// TIA Portal V16 export
// export: Created 2021-11-12T13:32:49.9949051Z, ExportSetting WithDefaults, DisplayName Totally Integrated Automation Portal, DisplayVersion V16 Update 3, DisplayName TIA Portal Version Control Interface, DisplayVersion V16 Update 2, DisplayName TIA Portal Openness, DisplayVersion V16 Update 3, DisplayName SINAMICS Startdrive Advanced, DisplayVersion V16 Update 5, DisplayName SINAMICS Startdrive G130, G150, S120, S150, SINAMICS MV, S210, DisplayVersion V16 Update 5, DisplayName SINAMICS Startdrive G110M, G120, G120C, G120D, G120P, G115D, DisplayVersion V16 Update 5, DisplayName STEP 7 Professional, DisplayVersion V16 Update 3, DisplayName STEP 7 Safety, DisplayVersion V16, DisplayName WinCC UA Professional, DisplayVersion V16 Update 3
DATA_BLOCK "HMI_CMD_310"   // DB70
{ S7_Optimized_Access := 'TRUE' }
VERSION : 0.1
// stored: AutoNumber true, DBAccessibleFromOPCUA true, IsOnlyStoredInLoadMemory false, IsRetainMemResEnabled false, IsWriteProtectedInAS false, MemoryReserve 100
   VAR
      xxxxx___BinarySensors___xxxxx_1 : Byte;
      "EQ01-BL01" : "UDT_CH_DI_Command";   // Sensor for min surface (LSL1444) / Hladina min (LSL1440)
      "EQ01-BL02" : "UDT_CH_DI_Command";   // Sensor for max surface (LSH 1445) / Hladina max (LSH 1441)
      "EQ01-BL03" : "UDT_CH_DI_Command";   // Level sensor Min LSL 1513 Pumping sump 2 (15m3) Level OK / Hladinový snímač Min LSL 1513 Čerpací jímka 2 (15m3) Hladina OK
      "EQ01-MA02_20" : "UDT_CH_DI_Command";   // Valve (A1419) - closed
      "EQ01-MA02_24" : "UDT_CH_DI_Command";   // Valve (A1419) - opened
      "EQ01-MA03_20" : "UDT_CH_DI_Command";   // Valve (A1416) - closed
      "EQ01-MA03_24" : "UDT_CH_DI_Command";   // Valve (A1416) - opened
      "EQ01-MA04_20" : "UDT_CH_DI_Command";   // Valve closed or in stroke (A1413)
      "EQ01-MA04_24" : "UDT_CH_DI_Command";   // Valve opened or in stroke (A1413)
      xxxxx___BinaryOthers___xxxxx_1 : Byte;
      "UC10-FC21_14" : "UDT_CH_DI_Command";   // 230V Hardening tube / 230V Zachlazovací nádrž
      "UC11-FC01_14" : "UDT_CH_DI_Command";   // 400V Pump of circulation P31 OK / 400V Čerpadlo cirkulace P31 OK
      DrainTank : Bool;   // Command to drain tank
      xxxxx___AnalogueSensors___xxxxx_1 : Byte;
      "EQ01-BT01" : "UDT_CH_AI_Command";   // Temperature measurment (TIC 1424) / Měření teploty (TIC 1424)
      "EQ01-BP01" : "UDT_CH_AI_Command";   // Tenzometric sond for measure surface (LIC 1430) / Tenzometrická sonda pro měření hladiny (LIC 1430)
      "EQ01-MA03_81" : "UDT_CH_AI_Command";   // Meření ventilu A 1416 Zavřeno - otevřeno
      xxxxx___Drives___xxxxx_1 : Byte;
      "EQ01-MA01" : "UDT_Drive1_Command";   // Pump of circulation (P31) / Čerpadlo cirkulace (P31)
      "EQ01-MA02" : "UDT_Valve2WB_Command";   // Valve with servomotor (A1419) - draining / Valve with servomotor (A1417) - draining
      "EQ01-MA03" : "UDT_Valve2WB_Command";   // Valve with servomotor (A1416) - cooling / Ventil se servopohonem (A1414) - chlazení
      "EQ01-MA04" : "UDT_Valve2WB_Command";   // Valve with servomotor (A1413) - filling / Ventil se servopohonem (A1411) - napouštění
      "UC11-TA01" : "UDT_SINAMICS_G120_Command";   // Frequence changer ( pro P33) / Frekvenční měnič ( pro P33)
      xxxxx___Alarms___xxxxx : Byte;
      ES : "UDT_DI_Mon_Command";   // E-stop
      KF31 : "UDT_DI_Mon_Command";   // module KF31
      Alarm_1 { S7_SetPoint := 'True'} : "UDT_DI_Mon_Command";   // Sensor Max level active and sensor Min level
      Alarm_2 { S7_SetPoint := 'True'} : "UDT_DI_Mon_Command";   // Sensor Min level active and analog level sensor under 10%
      Alarm_3 { S7_SetPoint := 'True'} : "UDT_DI_Mon_Command";   // Analog level sensor over 40% and sensor min level not active
      Alarm_4 { S7_SetPoint := 'True'} : "UDT_DI_Mon_Command";   // Water temperature high
      Alarm_5 { S7_SetPoint := 'True'} : "UDT_DI_Mon_Command";   // Water temperature low
      Alarm_6 { S7_SetPoint := 'True'} : "UDT_DI_Mon_Command";   // Water level high
      Alarm_7 { S7_SetPoint := 'True'} : "UDT_DI_Mon_Command";   // BSN3 tacts and water level NOK
      Alarm_8 { S7_SetPoint := 'True'} : "UDT_DI_Mon_Command";   // Filling and no water level change
      Alarm_9 { S7_SetPoint := 'True'} : "UDT_DI_Mon_Command";   // Drain and no water level change
   END_VAR
BEGIN
END_DATA_BLOCK
